{attribute 'qualified_only'}
{attribute 'strict'}
TYPE TriggerState :
(
	STOPPED, DELAY, ACTIVE_LOW, ACTIVE_HIGH
);
END_TYPE

(* stored: Version 1.1.0.1, ProductVersion 3.1.4024.15
   DUT TriggerState: Id {743077c5-5731-4fe8-b045-7b544d506422} *)
